FUNCTION_BLOCK PreExecutionChecks IMPLEMENTS I_PreExecutionChecks
VAR
	hasFailed : BOOL;
	hasFailedReason : T_MAXSTRING;
END_VAR;

METHOD PUBLIC Fail
VAR_INPUT
	Message : T_MAXSTRING;
END_VAR
IF hasFailed THEN
	RETURN;
END_IF

hasFailed := TRUE;
hasFailedReason := Message;
END_METHOD

PROPERTY PUBLIC Failed : BOOL
GET
Failed := hasFailed;
END_GET
END_PROPERTY

METHOD PUBLIC IsFalse
VAR_INPUT
	Actual : BOOL;
	Message : T_MAXSTRING;
END_VAR
IF hasFailed THEN
	RETURN;
END_IF

IF NOT Actual THEN
	RETURN;
END_IF

hasFailed := TRUE;
hasFailedReason := Message;
END_METHOD

METHOD PUBLIC IsTrue
VAR_INPUT
	Actual : BOOL;
	Message : T_MAXSTRING;
END_VAR
IF hasFailed THEN
	RETURN;
END_IF

IF Actual THEN
	RETURN;
END_IF

hasFailed := TRUE;
hasFailedReason := Message;
END_METHOD

PROPERTY PUBLIC Passed : BOOL
GET
Passed := not hasFailed;
END_GET
END_PROPERTY

PROPERTY PUBLIC Reason : T_MAXSTRING
GET
Reason := hasFailedReason;
END_GET
END_PROPERTY

METHOD PUBLIC Reset
VAR_INPUT
END_VAR
hasFailed := FALSE;
hasFailedReason := '';
END_METHOD

END_FUNCTION_BLOCK

(* stored: Version 1.1.0.1, ProductVersion 3.1.4024.15
   POU PreExecutionChecks: Id {95e3db63-eda6-05d0-1958-8e059c819b53}, SpecialFunc None
   Method Fail: Id {d1215c49-fb9b-02ce-3de6-a21e7bf14108}
   Property Failed: Id {38625ded-1fbf-0576-20fb-48fa61fa81a4}
   Get Get: Id {825a7bbc-fbb5-0f2f-2c60-48f2b199a5cc}
   Method IsFalse: Id {1353898e-74bb-0239-34ce-9683ff2879bc}
   Method IsTrue: Id {55fc693f-6c54-04af-083a-724685ca70c4}
   Property Passed: Id {d2f2e3bf-dddd-0afd-1476-90efc0ad65ca}
   Get Get: Id {d56e89c6-1f20-098e-3af4-7be030b64154}
   Property Reason: Id {67e2c1f0-1789-0a02-279a-8c115b90e613}
   Get Get: Id {920c4e1c-52dc-018e-0fda-d977d1813a45}
   Method Reset: Id {2be72906-41a7-04e9-39dd-1f3d59015f94} *)
